// TIA Portal V16 export
// export: Created 2021-11-12T13:32:44.1045203Z, ExportSetting WithDefaults, DisplayName Totally Integrated Automation Portal, DisplayVersion V16 Update 3, DisplayName TIA Portal Version Control Interface, DisplayVersion V16 Update 2, DisplayName TIA Portal Openness, DisplayVersion V16 Update 3, DisplayName SINAMICS Startdrive Advanced, DisplayVersion V16 Update 5, DisplayName SINAMICS Startdrive G130, G150, S120, S150, SINAMICS MV, S210, DisplayVersion V16 Update 5, DisplayName SINAMICS Startdrive G110M, G120, G120C, G120D, G120P, G115D, DisplayVersion V16 Update 5, DisplayName STEP 7 Professional, DisplayVersion V16 Update 3, DisplayName STEP 7 Safety, DisplayVersion V16, DisplayName WinCC UA Professional, DisplayVersion V16 Update 3
DATA_BLOCK "IDB_StationSCH1"   // DB170
{ DB_Accessible_From_OPC_UA := 'FALSE' }
VERSION : 0.1
// stored: AutoNumber true, DBAccessibleFromOPCUA false, InstanceOfName StationSCH1, InstanceOfType FB
"StationSCH1"
   // VAR_INPUT
   //    IS_Inputs : "UDT_COMM_SCH1_CRS";
   // END_VAR
   // VAR_OUTPUT
   //    OS_Outputs : "UDT_COMM_CRS_SCH1";
   //    OS_Status : "UDT_SCH_Status_specific";
   // END_VAR
   // VAR_IN_OUT
   //    XS_Parameter : "UDT_SCH_Parameter";
   //    XS_HMICommand : "UDT_SCH_Command";
   // END_VAR
   // VAR
   //    SF_Alarm1 : "STD_DI_Mon";
   //    SF_Alarm2 : "STD_DI_Mon";
   //    SF_Alarm3 : "STD_DI_Mon";
   //    SF_Alarm4 : "STD_DI_Mon";
   //    SF_Alarm5 : "STD_DI_Mon";
   //    SF_Alarm6 : "STD_DI_Mon";
   //    SF_Alarm7 : "STD_DI_Mon";
   //    SF_Alarm8 : "STD_DI_Mon";
   //    SF_Alarm9 : "STD_DI_Mon";
   //    SF_QW180 { S7_SetPoint := 'True'} : "STD_CH_AO";
   //    SF_QW182 { S7_SetPoint := 'True'} : "STD_CH_AO";
   //    SF_QW184 { S7_SetPoint := 'True'} : "STD_CH_AO";
   //    SF_QW186 { S7_SetPoint := 'True'} : "STD_CH_AO";
   //    Edge { S7_SetPoint := 'True'} : Array[0..31] of Bool;
   //    ST_Die3Rdy : TON_TIME;
   //    ST_Die456Rdy : TON_TIME;
   //    ST_StartPulse { S7_SetPoint := 'True'} : TP_TIME;
   // END_VAR
   // VAR RETAIN
   //    SDI_PartID : DInt;
   //    SI_PartType : Int;
   // END_VAR
   // VAR
   //    SF_Alarm10 { S7_SetPoint := 'True'} : "STD_DI_Mon";
   // END_VAR
BEGIN
END_DATA_BLOCK
